(*********************************** G.D S.p.A. - Technical Department ***********************************
============= PROGRAM INFO ============
FOLDER:             TBD
MACHINES INVOLVED:  TBD 

============= DESCRIPTION =============
csp machine declaration

============= REVISIONS ===============
Date		Version	 	Author      	Description             
----------	-------		------------  	--------------------------------------------
2019/04/05 	0000.00	 	M.Grasso		Creation of the PRG

**********************************************************************************************************)
(*$R process_ref := prc; $*)
PROGRAM csp_case_glue_ls_accU
VAR
	
	prc:											process;
	prc_path:										STRING;
	
END_VAR

_read_var_input();

_object_manager();

IF NOT objects_running()
THEN
	RETURN;	
END_IF

_read_process_image();

_mode_manager();

_set_runtime_properties();

(********************************* BODY *********************************)
(************************************************************************)

_handle_messages();

_write_output();

ACTION _handle_messages:
;
END_ACTION

ACTION _handle_process_test:
;
END_ACTION

ACTION _mode_manager:
IF process_mode_req_is_pending(prc)
THEN
    process_apply_mode_req_first_step(prc);
    CASE process_get_mode(prc) OF
        MODE_TO_ABSENT:
			;
        MODE_TO_INACTIVE:
			;
        MODE_TO_TEST:
			;
        MODE_TO_OPERATIONAL:
			;
    END_CASE
    process_apply_mode_req_second_step(prc);
END_IF
END_ACTION

ACTION _object_manager:
IF objects_initialization()
THEN
	sub_process_init(
		object_name					:= 'csp_case_glue_ls_accU.prc', 
		process						:= csp_case_glue_ls.prc, 
		CONVERSION_this				:= prc);
		
	prc_path 						:= process_get_path(prc);
END_IF

IF objects_running()
THEN
	process_cycle(prc);
END_IF
END_ACTION

ACTION _read_process_image:
;
END_ACTION

ACTION _read_var_input:
;
END_ACTION

ACTION _set_runtime_properties:
;
END_ACTION

ACTION _write_output:
;
END_ACTION

END_PROGRAM

(* stored: Version 1.1.0.1, ProductVersion 3.1.4022.12
   POU csp_case_glue_ls_accU: Id {c312d10f-d7b9-4d3d-aa6e-b6d9e149ad99}, SpecialFunc None
   Action _handle_messages: Id {de5cb4b6-5ee0-40fa-a74f-cb99c0b5dfb1}
   Action _handle_process_test: Id {f105282f-0922-421a-aff8-bf4ed1302da1}
   Action _mode_manager: Id {3991280c-3063-416d-9c86-866d6a7f9997}
   Action _object_manager: Id {94292e11-030d-418a-8491-6622ed6f608d}
   Action _read_process_image: Id {ca50427c-c564-49f2-b9f5-9df2c7d2335a}
   Action _read_var_input: Id {66fd9458-3921-4dc2-91b5-611e8fbc4068}
   Action _set_runtime_properties: Id {a09d09eb-ffe8-473a-9c3c-17863b41acbc}
   Action _write_output: Id {22d7c686-f34b-4610-ae05-74e2283a26fb} *)
